# EPICS autosave request: automation1App/Db/Automation1Hexapod_settings.req
$(P)$(H)Mode.VAL
$(P)$(H)MOVE_ALL_MODE.VAL
$(P)$(H)AUTO_TARGET_SYNC.VAL
$(P)$(H)TX.VAL
$(P)$(H)TY.VAL
$(P)$(H)TZ.VAL
$(P)$(H)TA.VAL
$(P)$(H)TB.VAL
$(P)$(H)TC.VAL
$(P)$(H)VEL.VAL
$(P)$(H)TX.PREC
$(P)$(H)TY.PREC
$(P)$(H)TZ.PREC
$(P)$(H)TA.PREC
$(P)$(H)TB.PREC
$(P)$(H)TC.PREC
$(P)$(H)VEL.PREC
